RoboDK station: Seguir_Trayectoria.rdk

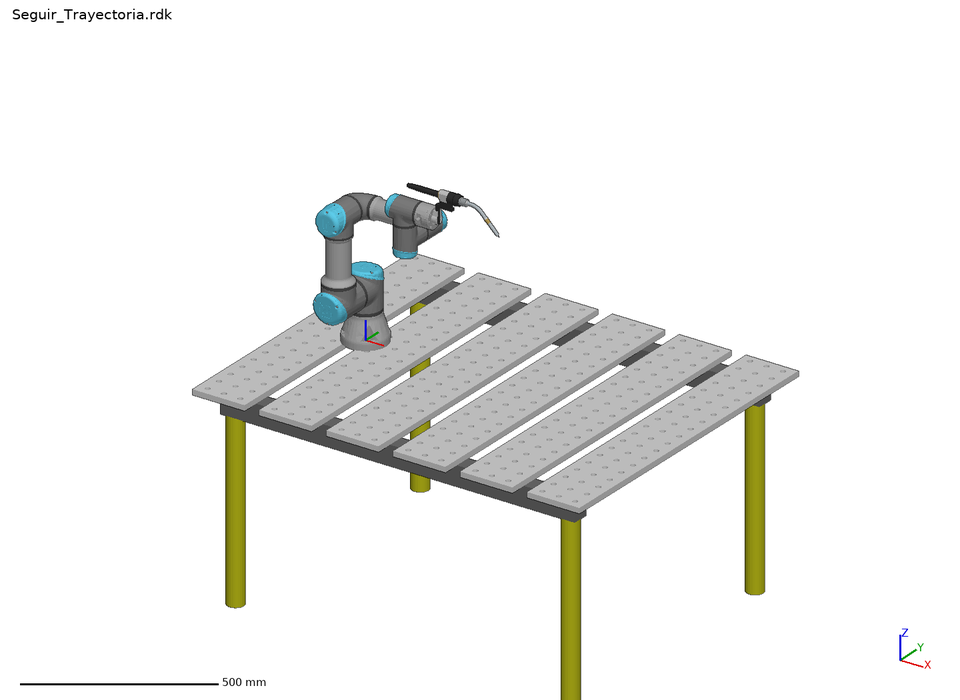
[picture v0: the station drawn from its stored meshes, robots at their saved joint values, targets as dots, program paths as lines]
Station Seguir_Trayectoria (saved by RoboDK 5.7.3). Poses are relative to the parent item; angles as X-Y-Z fixed-axis rotations.
  - frame UR3e Base at (-400, 0, 0) mm
    - robot UR3e: 6 axes, payload 3 kg, reach 500 mm, repeatability 0.03 mm, weight 11 kg
        modified DH rows (alpha deg, a mm, theta deg, d mm): 0, 0, 0, 151.9; 90, 0, 180, 0; 0, 243.55, 0, 0; 0, 213.2, 0, 131.05; -90, 0, 0, 85.35; 90, 0, 180, 92.1
        joint limits [-360, -360, -360, -360, -360, -360] to [360, 360, 360, 360, 360, 360]; home [0, -90, -90, 0, 90, 0]; saved at [0, -90, -90, 0, 90, 90]
      - tool OTC Daihen FD-84 Welding Gun, TCP at (1, 0, 201) mm, rotated rx 0 ry 45 rz 0 deg, size 100.8 x 32.5 x 283.9 mm
  - object Table 1200x1000mm (Welding) at (0, 0, 0) mm, size 1193.8 x 965.2 x 609.6 mm, geometry from Table-1200x1000mm-Welding.sld
